// TIA Portal V20 export
DATA_BLOCK "LBP_AlarmMsgs"   // DB2
TITLE = PLC-Error / Messages / Erreur AP / messages
{ S7_Optimized_Access := 'FALSE' }
AUTHOR : SINUMERIK
FAMILY : SINUMERIK_ONE
VERSION : 6.24
// Interface between user program and LBP_GenAlarmMsgs [FC10], contains bit arrays for blocking and stop signals as well as fault and status messages. / Interface entre programme utilisateur et LBP_GenAlarmMsgs [FC10] contient des tableaux de bits pour bloquer et arrêter des signaux et des signalisations de défaut et d'état.
// stored: AutoNumber false, InstanceOfName LBP_typeAlarmMsgs, InstanceOfType UDT
"LBP_typeAlarmMsgs"
   // VAR RETAIN
   //    Chan : Array[1..10] of Struct
   //       FDD : Array[0..15] of Bool;
   //       RID : Array[0..15] of Bool;
   //       NCSD : Array[0..15] of Bool;
   //       FdStop_1 : Array[0..15] of Bool;
   //       FdStop_2 : Array[0..15] of Bool;
   //       FdStop_3 : Array[0..15] of Bool;
   //    END_STRUCT;
   //    Axis : Array[1..31] of Struct
   //       FdStop : Array[0..15] of Bool;
   //    END_STRUCT;
   //    AddValUserA0 : Array[0..63] of Int;
   //    ChanA : Array[1..10] of Struct
   //       FDD_5C00xx : Array[0..15] of Bool;
   //       FDD_RID_5C01xx : Array[0..31] of Bool;
   //       RID_5C02xx : Array[0..31] of Bool;
   //       NCSD_5C03xx : Array[0..15] of Bool;
   //       FdStop_1_5C11xx : Array[0..15] of Bool;
   //       FdStop_2_5C12xx : Array[0..15] of Bool;
   //       FdStop_3_5C13xx : Array[0..15] of Bool;
   //    END_STRUCT;
   //    AxisA : Array[1..31] of Struct
   //       AAFdStop60AAxx : Array[0..15] of Bool;
   //    END_STRUCT;
   //    res552 : Word;
   //    UserA : Array[0..63] of Struct
   //       A70UUxx : Array[0..63] of Bool;
   //    END_STRUCT;
   // END_VAR
BEGIN
END_DATA_BLOCK
